(* PLC project  *)

CONFIGURATION FSOUT
END_CONFIGURATION
